//{{V2}}
ORGANIZATION_BLOCK OB1
TITLE= "Zyklisches Hauptprogramm"


AUTHOR:nb
FAMILY:nb
NAME:nb
VERSION:1.0


VAR_TEMP
       OB1_EV_CLASS:BYTE //Bits 0-3 = 1 (Coming event), Bits 4-7 = 1 (Event class 1)
       OB1_SCAN_1:BYTE //1 (Cold restart scan 1 of OB 1), 3 (Scan 2-n of OB 1)
       OB1_PRIORITY:BYTE //1 (Priority of 1 is lowest)
       OB1_OB_NUMBR:BYTE //1 (Organization block 1, OB1)
       OB1_RESERVED_1:BYTE //Reserved for system
       OB1_RESERVED_2:BYTE //Reserved for system
       OB1_PREV_CYCLE:INT //Cycle time of previous OB1 scan (milliseconds)
       OB1_MIN_CYCLE:INT //Minimum cycle time of OB1 (milliseconds)
       OB1_MAX_CYCLE:INT //Maximum cycle time of OB1 (milliseconds)
       OB1_DATE_TIME:DATE_AND_TIME //Date and time OB1 started
END_VAR
BEGIN

NETWORK
TITLE=
//{{a}}

//On reset do:
       UN   T         0
       SPBN _003

//calculate average of past values
       L    MW1004
       L    MW1002
       +I
       L    MW1000
       +I
       ITD
       DTR
       L    3.000000e+00
       /R
       T    MD2000


//shift values back
       L    MW1002
       T    MW1004

       L    MW1000
       T    MW1002

       L    0
       T    MW1000

_003:  NOP  0






//5s clock
       ON   T         0
       FP   M         0.0

       L    S5T#5S
       SV   T         0






//Zählen
       U    E         0.0
       FP   M         0.1
       SPBN _001

       L    1
       L    MW1000
       +I
       T    MW1000

_001:  NOP  1




//calculate speed and write to Output
       L    MD2000
       L    2.020000e+00
       *R
       L    5.000000e+00
       /R
       T    MD2004


       L    MD2004
       L    1.000000e+01
       *R
       RND
       ITB
       T    AW      100


       L    MD2004
       L    3.600000e+00
       *R
       T    MD2008

       L    MD2008
       L    1.000000e+01
       *R
       RND
       ITB
       T    AW      102
NETWORK
TITLE=
//{{a}}

       L    MD2008
       L    1.500000e+01
       >R
       SPBN _004
       L    1.500000e+01
       T    MD2008
_004:  NOP  0


       CALL FC      106
         IN:=MD2008
         HI_LIM:=1.500000e+01
         LO_LIM:=0.000000e+00
         BIPOLAR:=FALSE
         RET_VAL:=AW254
         OUT:=PAW256
END_ORGANIZATION_BLOCK
